TYPE (* Comma-separated list of communication profiles a device type supports (first entry is the default) *)
  (* Standard: 61499-1; Description: Copyright (c) 2026 Contributors to the Eclipse Foundation This program and the accompanying materials are made available under the terms of the Eclipse Public License 2.0 which is available at https://www.eclipse.org/legal/epl-2.0/ SPDX-License-Identifier: EPL-2.0 *)
  (* Version 1.0, 2026-07-17, Pedro Ricardo, initial API and implementation and/or initial documentation *)
  PACKAGE eclipse4diac::core;
  {SET_ATTRIBUTE(TARGET, (AutomationSystem:=FALSE,Application:=FALSE,GlobalConstant:=FALSE,Connection:=FALSE,Comment:=FALSE,Group:=FALSE,Link:=FALSE,ServiceSequence:=FALSE,FBType:=FALSE,SubAppType:=FALSE,DeviceType:=TRUE,ResourceType:=FALSE,SegmentType:=FALSE,DataType:=FALSE,AttributeDeclaration:=FALSE,FB:=FALSE,TypedSubApp:=FALSE,UntypedSubApp:=FALSE,Device:=FALSE,Resource:=FALSE,Segment:=FALSE,DataTypeMember:=FALSE,InstanceEvent:=FALSE,InstanceVarDecl:=FALSE,InstanceAdapter:=FALSE,TypeEvent:=FALSE,TypeVarDecl:=FALSE,TypeAdapter:=FALSE,Untyped_SubAppEvent:=FALSE,Untyped_SubAppVarDecl:=FALSE,Untyped_SubAppAdapter:=FALSE))}
  SupportedProfiles : STRING := ''; (* Comma-separated list of supported communication profiles (first entry is the default) *)
END_TYPE
